FUNCTION_BLOCK FB_ejemplo_Method
VAR_INPUT
END_VAR
VAR_OUTPUT
END_VAR
VAR
	bBool : BOOL;
	ststruct : ST_sample2;
	fb5 : fbreturn5;
END_VAR

METHOD metodo1_a_Cero_bBool
THIS^.bBool := false;
END_METHOD

METHOD metodo1_a_Cero_InOut : bool
VAR_IN_OUT
	bBool : BOOL;
END_VAR
// Método que pone a 0 la variable definida en in_Out
bBool := FALSE;
// return value bBOOL
metodo1_a_Cero_InOut := FALSE;
END_METHOD

METHOD metodo1_a_Uno_bBool
THIS^.bBool := true;
END_METHOD

METHOD metodo1_a_Uno_InOut : BOOL
VAR_IN_OUT
	bBool : BOOL;
END_VAR
// Método que pone a 1 la variable definida en in_Out
bBool := TRUE;
// return value bBOOL
metodo1_a_Uno_InOut := TRUE;
END_METHOD

METHOD PUBLIC metodo2_struct : REFERENCE TO ST_sample2
VAR_INPUT
	st_struct : ST_sample2;
END_VAR


THIS^.ststruct := st_struct;

metodo2_struct REF= THIS^.ststruct;
END_METHOD

METHOD PRIVATE metodo3_interface : interface3
VAR_INPUT
END_VAR
END_METHOD

METHOD Metodo4_VarInst : INT
VAR_OUTPUT
	outvarcounter : INT;
END_VAR
VAR
	varcounter : INT;
END_VAR
VAR_INST
	counter : INT;
END_VAR
counter := counter + 1;
Metodo4_VarInst := counter;

varcounter := varcounter + 1; 
outvarcounter := varcounter;
END_METHOD

METHOD metodo5_returnfb : fbreturn5
VAR_INPUT
END_VAR
metodo5_returnfb := fb5;
END_METHOD

END_FUNCTION_BLOCK

(* stored: Version 1.1.0.1, ProductVersion 3.1.4024.12
   POU FB_ejemplo_Method: Id {bf742efc-6283-4256-8c15-fe1e5052c0b1}, SpecialFunc None
   Method metodo1_a_Cero_bBool: Id {8e330d49-1f63-4334-814e-68871791412a}
   Method metodo1_a_Cero_InOut: Id {ca391e3d-beb1-4763-9e11-9b19da417c6f}
   Method metodo1_a_Uno_bBool: Id {a0dd2c9e-b6be-44bf-82f5-91ed7c375ad6}
   Method metodo1_a_Uno_InOut: Id {a76f9dae-a442-4326-8bff-bcdcbcef124c}
   Method metodo2_struct: Id {72fb7591-8743-4488-8a14-c4c09928a599}
   Method metodo3_interface: Id {709f3c2b-aebf-4e82-82e6-70b51bb45770}
   Method Metodo4_VarInst: Id {3461a640-013c-4a20-bed4-dff49f316726}
   Method metodo5_returnfb: Id {bf88f70d-1d25-4abb-b32e-abebdb5103db} *)
